# EPICS autosave request: galilDmc30017App/Db/galil_dmc30017_analog_out.req
# The files listed here are located at <GALIL support top>/GalilSup/Db
# as they are provided by the Galil Support Module

# All 2 Analog outputs
file "galil_analog_out.req" P=$(P), R=$(ANALOG_OUT0)
file "galil_analog_out.req" P=$(P), R=$(ANALOG_OUT1)
